(* IEC 61131-3 sources: robocpp/validation/corpus/accepted, 2 files *)

(* ---- counter.st ---- *)
(* validation: feature=language.st clause=3.3 *)
PROGRAM CounterDemo
VAR
    Count : INT := 0;
    Limit : INT := 3;
    Done : BOOL := FALSE;
END_VAR

IF Count < Limit THEN
    Count := Count + 1;
ELSE
    Done := TRUE;
END_IF;
END_PROGRAM

(* ---- instruction_list.il ---- *)
(* validation: feature=language.il clause=3.2 *)
PROGRAM InstructionListFile
VAR
    A : INT := 3;
    B : INT := 4;
    Sum : INT := 0;
    Bigger : BOOL := FALSE;
END_VAR

LD A
ADD B
ST Sum
LD Sum
GT 5
ST Bigger
END_PROGRAM
